PROGRAM MAIN
VAR
	fbModule1:		FB_Module01;	
	bReset:			BOOL;
	bStart: 		BOOL;
    bHold:       	BOOL;
    bPause:    		BOOL;
	bStop:       	BOOL;
    bAbort:      	BOOL;

END_VAR


fbModule1();

IF bReset THEN
	bReset:= NOT fbModule1.M_Request(E_Request.Reset);
END_IF

IF bStart THEN
	bStart:= NOT fbModule1.M_Request(E_Request.Start);
END_IF

IF bStop THEN
	bStop:= fbModule1.M_Request(E_Request.Stop);
END_IF

IF bHold THEN
	bHold:= NOT fbModule1.M_Request(E_Request.Hold);
END_IF

IF bPause THEN
	bPause:= NOT fbModule1.M_Request(E_Request.Pause);
END_IF

IF bAbort THEN
	bAbort:= NOT fbModule1.M_Request(E_Request.Abort);
END_IF

END_PROGRAM

(* stored: Version 1.1.0.1, ProductVersion 3.1.4024.12
   POU MAIN: Id {80fd576e-8bda-0001-19b1-22d89fc11873}, SpecialFunc None *)
